VAR_GLOBAL
(*
    Only includes motor definitions for the IOC
    These are hard-coded to be Main.M#,
    but are very convenient to store in a GVL,
    hence the confusing namespace here

    This should be refactored once the IOC
    supports arbitrary ads paths for motors
*)
    (*DCCM Mono*)
    // Motors
	                                               
    {attribute 'TcLinkTo' := '.bLimitForwardEnable:=TIID^Device 2 (EtherCAT)^EK1200_DCCM^EL7047_DCCM_th1^STM Status^Status^Digital input 1;
                              .bLimitBackwardEnable:=TIID^Device 2 (EtherCAT)^EK1200_DCCM^EL7047_DCCM_th1^STM Status^Status^Digital input 2;'}
    {attribute 'pytmc' := '
        pv: DCCM:SWITCH:MMS:TH1
    '}
    M1 : DUT_MotionStage := (fVelocity:=100.0, nEnableMode:=ENUM_StageEnableMode.ALWAYS, bPowerSelf:=TRUE); // DCCM th1
    fbMotionStage_m1 : FB_MotionStage;

    {attribute 'TcLinkTo' := '.bLimitForwardEnable:=TIID^Device 2 (EtherCAT)^EK1200_DCCM^EL7047_DCCM_th2^STM Status^Status^Digital input 1;
                              .bLimitBackwardEnable:=TIID^Device 2 (EtherCAT)^EK1200_DCCM^EL7047_DCCM_th2^STM Status^Status^Digital input 2;'}
    {attribute 'pytmc' := '
        pv: DCCM:SWITCH:MMS:TH2
    '}
    M2 : DUT_MotionStage := (fVelocity:=100.0, nEnableMode:=ENUM_StageEnableMode.ALWAYS, bPowerSelf:=TRUE); // DCCM th2
    fbMotionStage_m2 : FB_MotionStage;

	{attribute 'TcLinkTo' := '.bLimitForwardEnable:=TIID^Device 2 (EtherCAT)^EK1200_DCCM^EL7047_DCCM_tx^STM Status^Status^Digital input 1;
                              .bLimitBackwardEnable:=TIID^Device 2 (EtherCAT)^EK1200_DCCM^EL7047_DCCM_tx^STM Status^Status^Digital input 2;'}
    {attribute 'pytmc' := '
        pv: DCCM:SWITCH:MMS:TX
    '}
    M3 : DUT_MotionStage := (fVelocity:=150.0, nEnableMode:=ENUM_StageEnableMode.ALWAYS, bPowerSelf:=TRUE); // DCCM tx
    fbMotionStage_m3 : FB_MotionStage;

    {attribute 'TcLinkTo' := '.bLimitForwardEnable:=TIID^Device 2 (EtherCAT)^EK1200_DCCM^EL7047_DCCM_txd^STM Status^Status^Digital input 1;
                              .bLimitBackwardEnable:=TIID^Device 2 (EtherCAT)^EK1200_DCCM^EL7047_DCCM_txd^STM Status^Status^Digital input 2;'}
    {attribute 'pytmc' := '
        pv: DCCM:SWITCH:MMS:TXD
    '}
    M4 : DUT_MotionStage := (fVelocity:=150.0, nEnableMode:=ENUM_StageEnableMode.ALWAYS, bPowerSelf:=TRUE); // DCCM txd
    fbMotionStage_m4 : FB_MotionStage;

    {attribute 'TcLinkTo' := '.bLimitForwardEnable:=TIID^Device 2 (EtherCAT)^EK1200_DCCM^EL7047_DCCM_txy^STM Status^Status^Digital input 1;
                              .bLimitBackwardEnable:=TIID^Device 2 (EtherCAT)^EK1200_DCCM^EL7047_DCCM_txy^STM Status^Status^Digital input 2;'}
    {attribute 'pytmc' := '
        pv: DCCM:SWITCH:MMS:txy
    '}
    M5 : DUT_MotionStage := (fVelocity:=30.0, nEnableMode:=ENUM_StageEnableMode.DURING_MOTION, bPowerSelf:=TRUE); // DCCM txy
	fbMotionStage_m5 : FB_MotionStage;	
	
	M1_encoder : DUT_MotionStage := (fVelocity:=100.0, nEnableMode:=ENUM_StageEnableMode.ALWAYS, bPowerSelf:=TRUE); // DCCM th1 encoder
    fbMotionStage_m1_encoder : FB_MotionStage;

 	M2_encoder : DUT_MotionStage := (fVelocity:=100.0, nEnableMode:=ENUM_StageEnableMode.ALWAYS, bPowerSelf:=TRUE); // DCCM th2 encoder
    fbMotionStage_m2_encoder : FB_MotionStage;
	
	M3_encoder : DUT_MotionStage := (fVelocity:=100.0, nEnableMode:=ENUM_StageEnableMode.ALWAYS, bPowerSelf:=TRUE); // DCCM tx encoder
     fbMotionStage_m3_encoder : FB_MotionStage;
	
	M4_encoder : DUT_MotionStage := (fVelocity:=100.0, nEnableMode:=ENUM_StageEnableMode.ALWAYS, bPowerSelf:=TRUE); // DCCM tx_d encoder
     fbMotionStage_m4_encoder : FB_MotionStage;
	
	M5_encoder : DUT_MotionStage := (fVelocity:=100.0, nEnableMode:=ENUM_StageEnableMode.ALWAYS, bPowerSelf:=TRUE); // DCCM ty_d encoder
     fbMotionStage_m5_encoder : FB_MotionStage;
END_VAR

(* stored: Version 1.1.0.1, ProductVersion 3.1.4024.12
   GVL Main: Id {70c05a97-6edf-41f6-937c-0e62f3a09f50} *)
